// TIA Portal V16 export
// export: Created 2023-09-11T12:14:55.8710509Z, ExportSetting WithDefaults, DisplayName Totally Integrated Automation Portal, DisplayVersion V16 Update 6, DisplayName TIA Portal Version Control Interface, DisplayVersion V16 Update 2, DisplayName TIA Portal Openness, DisplayVersion V16 Update 6, DisplayName STEP 7 Professional, DisplayVersion V16 Update 6, DisplayName STEP 7 Safety, DisplayVersion V16, DisplayName WinCC Advanced, DisplayVersion V16 Update 6
DATA_BLOCK "db10datablock"   // DB10
TITLE = Instance SCADA
{ S7_Optimized_Access := 'FALSE' }
AUTHOR : RTecmer
VERSION : 0.1
// stored: AutoNumber false, DBAccessibleFromOPCUA true, IsOnlyStoredInLoadMemory false, IsWriteProtectedInAS false
   VAR
      Clock : Time;
      Watchdog : Int;
      State_6 : Word;
      State_7 : Word;
      State_8 : Word;
      State_9 : Word;
      State_10 : Real;
      State_11 : Real;
      State_12 : Word;
      State_13 : Word;
      State_14 : DWord;
      State_15 : DWord;
      State_16 : DWord;
      State_17 : DWord;
      State_18 : Int;
      State_19 : Int;
      State_20 : Int;
      State_21 : Int;
      State_22 : Int;
      State_23 : Real := 2.2;
      State_24 : Real := 1.5;
      State_25 : Real;
      setpoint_SV_bar : Real := 1.8;   // Zadana wartość ciśnienie do PID [bar]
      State_26 : Real := 0.0;
      instFlowDN225_act_Q1 : Real;   // aktualny przepływ Q1 pompownia
      reset_modbus_TCP : Bool;   // reset komunikacji modbus TCP
      instB7_bar_act_pompownia : Real := 0.28;   // aktualne
      State_27 : Real := 1.7;
      State_28 : Real := 2.7;
      State_90 : Real;   // aktualny czas
      State_29 : Real;
      act_stanP1 : Int;   // Zmienna na potzrzeby trenów pracy pompy
      act_statnP2 : Int;   // Zmienna na potzrzeby trenów pracy pompy
      act_stanP3 : Int;   // Zmienna na potzrzeby trenów pracy pompy
      act_stanP4 : Int;
      instSumFlowDN225_Q1 : Real;   // Aktualny przepływ na wlocie oczyszczalni m3/h
      State_30 : Word := 1;
      State_31 : Real;
      "alarms only" : Word;   // Instancja alarmów (bit 146.4 - Error Modbus),(bit 146.5-Warning Modbau)
      inverterPomp_Status : Word;   // Status falownika pomp
      inst_act_Current_Inverters : Real;   // Aktualny prąd falownika [A]
      set_press_bar_Max : Real := 7.888;   // Maxymalne dopuszczalne ciśnienie w rurociągu [bar]
      State_128 : Real := 56.0;
      act_Hz_Inverter_1 : Real;   // Aktualne Hz na falowniku
      ins_ModeWorkContactronP1 : Word;   // Zmienna przechowująca informację o stanie napędu (0-postój, 1-falownik, 2-sieć)
      ins_ModeWorkContactronP2 : Word;   // Zmienna przechowująca informację o stanie napędu (0-postój, 1-falownik, 2-sieć)
      ins_ModeWorkContactronP3 : Word;   // Zmienna przechowująca informację o stanie napędu (0-postój, 1-falownik, 2-sieć)
      ins_ModeWorkContactronP4 : Word;   // Zmienna przechowująca informację o stanie napędu (0-postój, 1-falownik, 2-sieć)
      instB9_bar_act_Granica : Real;   // Wartość bar w sterowanym zbiorniku
      PV_HWrn_set_correct : Real := 2.1;   // Wspóczninik służący wprowadzeniu korekty ostrzeżenia przekroczenia wartości zadanej bar
      PV_LWrn_set_correct : Real := 0.6;   // Wspóczninik służący wprowadzeniu korekty ostrzeżenia zbyt niskia wartości bar w stosunku do zadanej
      TimeHistere_set_bar : Int := 1;   // Czas zwłoki przed zmianą bar zadanego podczas redukcji azotu
      avg_bar : Real;   // srednia wartość ciśnienie
      RTU_Fal_1errorStatus : Word;   // Status błędu komunikacji Modbus RTU
      RTU_MPP04_1errorStatus : Word;   // Status błędu komunikacji Modbus RTU
      RTU_MPP04_2errorStatus : Word;   // Status błędu komunikacji Modbus RTU
      RTU_MT101 : Word;   // Status błędu komunikacji Modbus RTU
      RTU_stepRESET : Bool := 1;   // Krok pętli Modbus RTU na potrzeby SCADA (RESET)
      setRTU_Error : Bool;   // Znacznik błedu modbus RTU
      instSecStart_City_1 : Int;   // Sekundy start przetłaczanie
      instSecStop_City_1 : Int;   // Sekundy stop przetłaczanie
      instSecStart_Replen_1 : Int;   // Sekundy start dosilanie
      instSecStop_Replen_1 : Int;   // Sekundy stop dosilanie
      CounterOverTempFa : Int;   // Licznik wystąpienia usterki przegrzania
      instSecStart_Filling_1 : Int;   // Sekundy start napełniania
      instSecStop_Filling_1 : Int;   // Sekundy stop napełniania
      CounterOverVoltFal : Int;   // Licznik wystapienia usterki wysokie VDC
      instHourStart_Filling_1 : Int;   // Godzina start napełniania
      instMinutStart_Filling : Int;   // Minuta start napełniania
      instHourStop_Filling_1 : Int;   // Godzina stop napełniania
      instMinutStopt_Filling : Int;   // Minuta stop napełniania
      instFlowDN500_act_Q2 : Real;   // Aktualna wartośc przepływu Q2 magistrala
      instSumFlowDN500_Q2 : Real;   // Aktualna wartośc sumy przepywu Q2 magistrala
      instHourStart_Filling : DTL;   // Godzina start napełniania
      instHourStop_Filling : DTL;   // Godzina stop napełniania
      instHourStart_City : DTL;   // Godzina start przetłaczanie miasto DN225
      instHourStop_City : DTL;   // Godzina stop przetłaczanie miasto DN225
      instHourStart_Replen : DTL;   // Godzina start dosilanie DN500
      instHourStop_Replen : DTL;   // Godzina stop dosilanie DN500
      actQ1_przepyw_pompownia_Int : Word;   // Aktualny przepływ na Q1 pompownia
      actQ2_przepyw_pompownia_Int : Word;   // Aktualny przepływ na Q2 pompownia
      inst_sum_FlowDN255_act_Q2_int : Word;   // aktualna suma przepływu Q1 (int)
      inst_sumFlowDN500_act_Q2_int : Word;   // aktualna suma przepływu Q2 (int)
      instHourStart_City_1 : Int;   // Godzina start przetłaczanie miasto DN225
      instMinutStart_City : Int;   // Minuty start przetłaczanie miasto DN225
      instHourStop_City_1 : Int;   // Godzina stop przetłaczanie miasto DN225
      instMinutStopt_City : Int;   // Minuty stop przetłaczanie miasto DN225
      instHourStart_Replen_1 : Int;   // Godzina start dosilanie magistrala DN500
      instMinutStart_Replen : Int;   // Minuty start dosilanie magistrala DN500
      instHourStop_Replen_1 : Int;   // Godzina stop dosilanie magistrala DN500
      instMinutStopt_Replen : Int;   // Minuty stop dosilanie magistrala DN500
      instvValveZ1 : Word;   // Zasuwa zbiornik - spust zbiornik 1
      instvValveZ2 : Word;   // Zasuwa zbiornik - zasilanie zbiornik 1
      instvValveZ3 : Word;   // Zasuwa zbiornik - spust zbiornik 2
      instvValveZ4 : Word;   // Zasuwa zbiornik - zasilanie zbiornik 2
      instvValveZ5 : Word;   // Zasuwa zbiornik - spust zbiornik 3
      instvValveZ6 : Word;   // Zasuwa zbiornik - zasilanie zbiornik 3
      instvValveZ7 : Word;   // Zasuwa zbiornik - spust zbiornik 4
      instvValveZ8 : Word;   // Zasuwa zbiornik - zasilanie zbiornik 4
      instvValveZ9 : Word;   // Zasuwa suchobieg
      instvValveZ10 : Word;   // Zasuwa zbiornik regulowana - zasilanie
      actHour : Int;   // Godzina start dosilanie magistrala DN500
      actMinut : Int;   // aktualny czas
      actSec : Int := 0;   // aktualny czas
      Time_ONK3 : Int := 45;   // timer na on pompy dodatkowej
      Time_OFFK3 : Int := 2;   // timer na off pompy dodatkowej
      received_zero { S7_SetPoint := 'True'} : "typeDataInverter_Word";   // wielkość przepływu
      received_zero_1 { S7_SetPoint := 'True'} : "typeDataInverter_DWord";   // Podwójne słowo czasu pracy falownika [Int32, index -0]
      received_zero_2 { S7_SetPoint := 'True'} : "typeDataInverter_Word";   // Podwójne słowo czasu pracy falownika [Int32, index -0]
   END_VAR
BEGIN
   received_zero.typeDataInverter_int[0] := 0;
   received_zero_1.typeDataInverter_Dword[0] := 0;
   received_zero_2.typeDataInverter_int[0] := 0;
END_DATA_BLOCK
